PROGRAM Voyants
VAR // added by the converter: edge detectors and wires of the graphical bodies
    _w1, _w2, _w3 : BOOL;
END_VAR

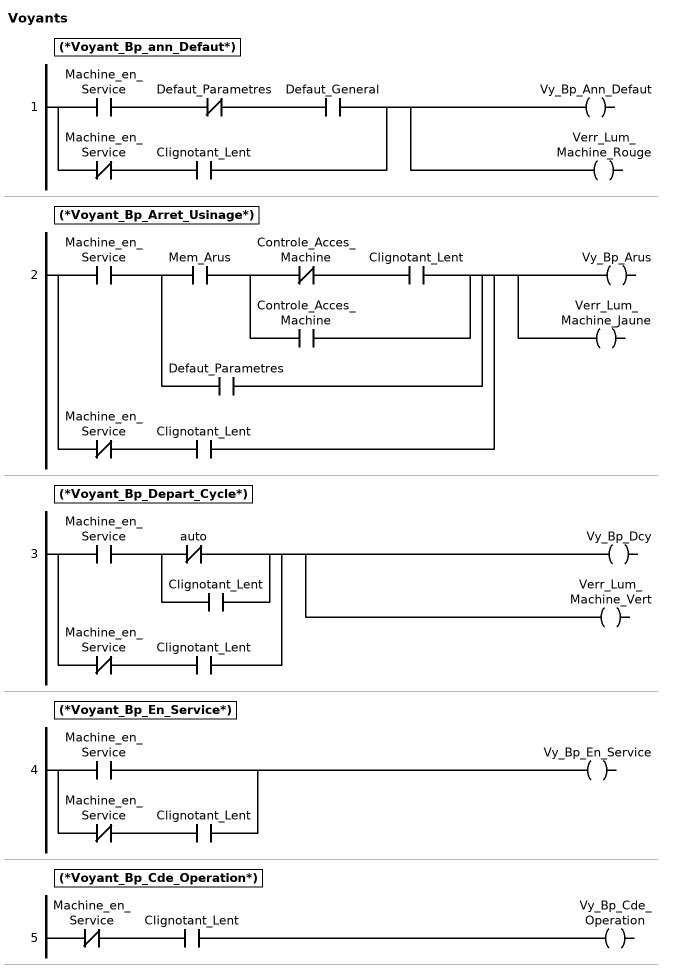
// NETWORK 1
// label: (*Voyant_Bp_ann_Defaut*)
_w1 := Machine_en_Service AND NOT Defaut_Parametres AND Defaut_General OR NOT Machine_en_Service AND Clignotant_Lent;
Vy_Bp_Ann_Defaut := _w1;
Verr_Lum_Machine_Rouge := _w1;

// NETWORK 2
// label: (*Voyant_Bp_Arret_Usinage*)
_w2 := Machine_en_Service AND (Mem_Arus AND (NOT Controle_Acces_Machine AND Clignotant_Lent OR Controle_Acces_Machine) OR Defaut_Parametres) OR NOT Machine_en_Service AND Clignotant_Lent;
Vy_Bp_Arus := _w2;
Verr_Lum_Machine_Jaune := _w2;

// NETWORK 3
// label: (*Voyant_Bp_Depart_Cycle*)
_w3 := Machine_en_Service AND (NOT auto OR Clignotant_Lent) OR NOT Machine_en_Service AND Clignotant_Lent;
Vy_Bp_Dcy := _w3;
Verr_Lum_Machine_Vert := _w3;

// NETWORK 4
// label: (*Voyant_Bp_En_Service*)
Vy_Bp_En_Service := Machine_en_Service OR NOT Machine_en_Service AND Clignotant_Lent;

// NETWORK 5
// label: (*Voyant_Bp_Cde_Operation*)
Vy_Bp_Cde_Operation := NOT Machine_en_Service AND Clignotant_Lent;

END_PROGRAM

(* stored: Version 1.1.0.1
   POU Voyants: Id {63a91442-01fd-46b9-9a17-4798b77d9843}, SpecialFunc None *)
